// TIA Portal project "P8_sim_v2" (V14)

(* hardware
DEVICE "S7-1200 station_1"  S7-1200 Station
   slot 0: "Rack_0"  S7-1200 Rack  Rack  V1.0
   slot 1: "PLC_1"  CPU 1214C AC/DC/Rly  6ES7 214-1BG40-0XB0  V4.2
*)

// ===== PLC "PLC_1"  CPU 1214C AC/DC/Rly =====

VAR_GLOBAL   // PLC tag table "Default tag table"
   ""PM"" AT %I0.0 : Bool;
   ""PP"" AT %I0.1 : Bool;
   ""FCA_1"" AT %I0.2 : Bool;
   ""FCB_1"" AT %I0.3 : Bool;
   ""CW_1"" AT %Q0.0 : Bool;
   ""CCW_1"" AT %Q0.1 : Bool;
END_VAR